TYPE T_ASTRO_MEAN_COORDINATES :
STRUCT
	alpha : 	LREAL := 0.0;
	delta : 	LREAL := -890000.0;
	epoch : 	LREAL;
	equinox : 	LREAL := 2000;
	pma : 		LREAL;
	pmd : 		LREAL;
	radvel : 	LREAL;
	parallax : 	LREAL;
END_STRUCT
END_TYPE

(* stored: Version 1.1.0.1, ProductVersion 3.1.4024.11
   DUT T_ASTRO_MEAN_COORDINATES: Id {cac6d104-11fa-49b5-8871-ae9133e2acbd} *)
